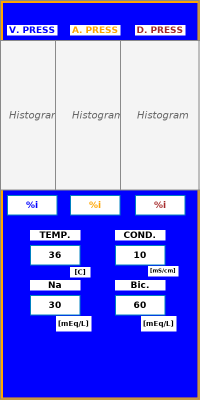
VISUALIZATION Data_Left  // 200x400
    Rectangle (0,0 200x400)
    Histogram (-8,40 86x150), scale format: %1.1f, scale -100..300
        p518627256: mmHg
        p1518820177: HMI_Global.HMI_ArrayGraph1
        p102497268: HMI_Global.HMI_ArrayGraph1
        p788070771: ARRAY [0..1] OF INT
    Histogram (55,40 86x150), scale format: %1.1f, scale -300..100
        p518627256: mmHg
        p1518820177: HMI_Global.HMI_ArrayGraph2
        p102497268: HMI_Global.HMI_ArrayGraph2
        p788070771: ARRAY [0..1] OF INT
    Histogram (120,40 86x150), scale format: %1.1f, scale -400..300
        p518627256: mmHg
        p1518820177: HMI_Global.HMI_ArrayGraph3
        p102497268: HMI_Global.HMI_ArrayGraph3
        p788070771: ARRAY [0..1] OF INT
    Textfield (7,25 50x10), "V. PRESS"
    Textfield (70,25 50x10), "A. PRESS"
    Textfield (135,25 50x10), "D. PRESS"
    Textfield (7,195 50x20), "%i"
    Textfield (70,195 50x20), "%i"
    Textfield (135,195 50x20), "%i"
    Textfield (30,245 50x20), "36"
    Textfield (115,295 50x20), "60"
    Textfield (115,245 50x20), "10"
    Textfield (30,295 50x20), "30"
    Textfield (30,230 50x10), "TEMP."
    Textfield (115,230 50x10), "COND."
    Textfield (115,280 50x10), "Bic."
    Textfield (30,280 50x10), "Na"
    Textfield (70,267 20x10), "[C]"
    Textfield (148,266 30x10), "[mS/cm]"
    Textfield (56,316 35x15), "[mEq/L]"
    Textfield (141,316 35x15), "[mEq/L]"
END_VISUALIZATION

(* stored: Version 1.1.0.1, ProductVersion 3.1.4024.12
   Visu Data_Left: Id {8d398a51-fee6-4abc-9ca3-0795414f09cd} *)
